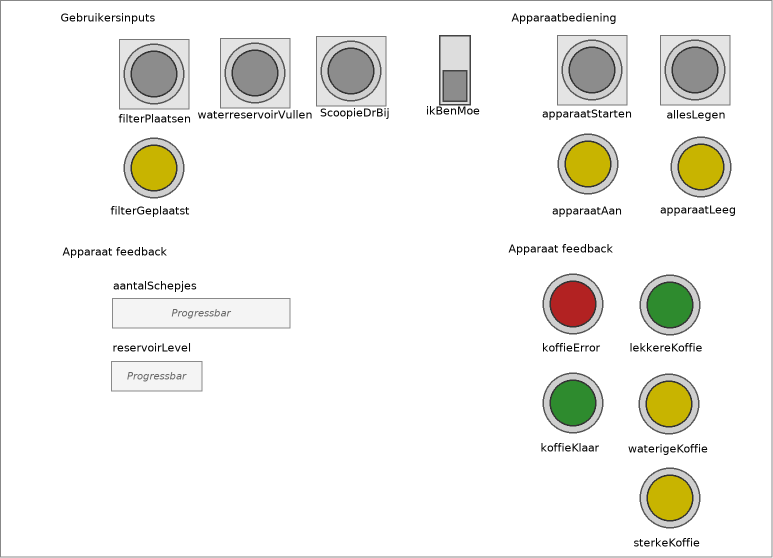
VISUALIZATION Visualization  // 773x558
    Lamp1 (553,129 70x70), variable: MAIN.apparaatAan, style: Lamp-Lamp1-Yellow
    Lamp1 (119,133 70x70), variable: MAIN.filterGeplaatst, style: Lamp-Lamp1-Yellow
    Lamp1 (538,368 70x70), variable: MAIN.koffieKlaar, style: Lamp-Lamp1-Green
    Lamp1 (538,269 70x70), variable: MAIN.koffieError, style: Lamp-Lamp1-Red
    Lamp1 (666,132 70x70), variable: MAIN.apparaatLeeg, style: Lamp-Lamp1-Yellow
    Label (512,99 150x30), "apparaatStarten"
    Label (512,196 150x30), "apparaatAan"
    Label (623,195 150x30), "apparaatLeeg"
    Label (495,433 150x30), "koffieKlaar"
    Label (496,333 150x30), "koffieError"
    Label (75,196 150x30), "filterGeplaatst"
    Label (80,104 150x30), "filterPlaatsen"
    Label (180,100 150x30), "waterreservoirVullen"
    Label (280,98 150x30), "ScoopieDrBij"
    Label (621,100 150x30), "allesLegen"
    DipSwitch (420,35 70x70), variable: MAIN.ikBenMoe, behaviour: TOGGLE, style: Switch-DipSwitch-Gray
    Label (378,96 150x30), "ikBenMoe"
    Lamp1 (635,270 70x70), variable: MAIN.lekkereKoffie, style: Lamp-Lamp1-Green
    Lamp1 (635,463 70x70), variable: MAIN.sterkeKoffie, style: Lamp-Lamp1-Yellow
    Lamp1 (634,369 70x70), variable: MAIN.waterigeKoffie, style: Lamp-Lamp1-Yellow
    Label (592,528 150x30), "sterkeKoffie"
    Label (593,434 150x30), "waterigeKoffie"
    Label (591,333 150x30), "lekkereKoffie"
    Label (80,271 150x30), "aantalSchepjes"
    Label (77,333 150x30), "reservoirLevel"
    PushSwitch (119,39 70x70), variable: GVL.filterPlaatsen, behaviour: TAP, style: Switch-PushSwitch-Gray
    PushSwitch (220,38 70x70), variable: GVL.waterreservoirVullen, behaviour: TAP, style: Switch-PushSwitch-Gray
    PushSwitch (316,36 70x70), variable: GVL.scoopieDrBij, behaviour: TAP, style: Switch-PushSwitch-Gray
    PushSwitch (660,35 70x70), variable: GVL.allesLegen, behaviour: TAP, style: Switch-PushSwitch-Gray
    PushSwitch (557,35 70x70), variable: GVL.apparaatAanzetten, behaviour: TAP, style: Switch-PushSwitch-Gray
    Progressbar (112,298 178x30), variable: aantalSchepjes
    Label (33,3 150x30), "Gebruikersinputs"
    Label (40,237 150x30), "Apparaat feedback"
    Progressbar (111,361 91x30), variable: reservoirLevel
    Label (489,3 150x30), "Apparaatbediening"
    Label (486,234 150x30), "Apparaat feedback"
END_VISUALIZATION

(* stored: Version 1.1.0.1, ProductVersion 3.1.4024.12
   Visu Visualization: Id {9d4f1e3d-2e67-4bc5-8272-0d646e0dfaa8} *)
